TYPE ST_AKcabinetPanel :
STRUCT
	inputs : ST_AKcabinetPanelInputs;
	outputs : ST_AKcabinetPanelOutputs;
END_STRUCT
END_TYPE

(* stored: Version 1.1.0.1, ProductVersion 3.1.4024.4
   DUT ST_AKcabinetPanel: Id {6616af60-27a9-49e0-9046-153de74d854d} *)
